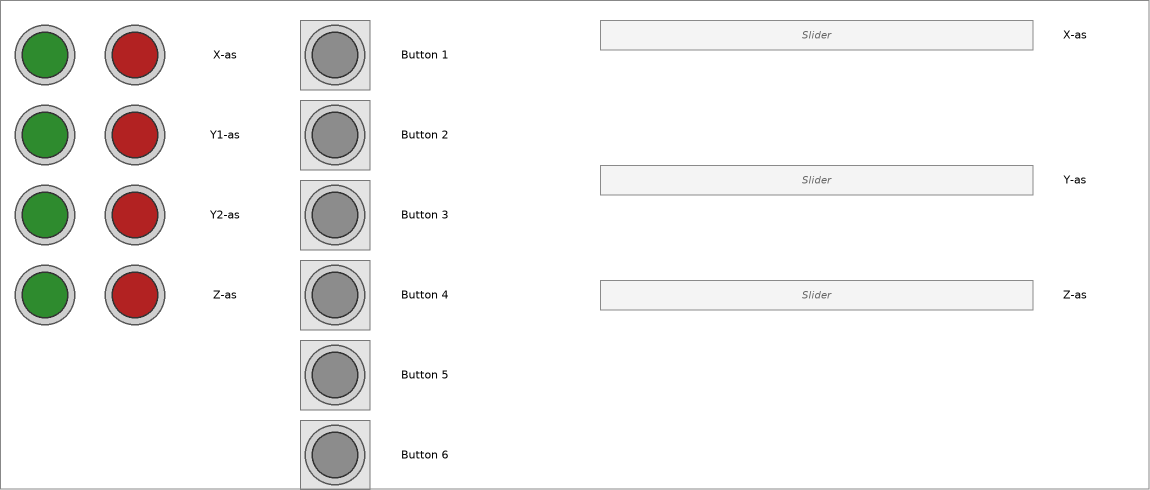
VISUALIZATION Visu  // 1150x490
    Slider (600,20 433x30), variable: GVL.slider1, scale 25..375
    Slider (600,165 433x30), variable: GVL.slider2, scale 25..375
    Slider (600,280 433x30), variable: GVL.slider3, scale 25..125
    Lamp1 (100,20 70x70), variable: GVL.bLed_Rd1, style: Lamp-Lamp1-Red
    Lamp1 (100,260 70x70), variable: GVL.bLed_Rd4, style: Lamp-Lamp1-Red
    Lamp1 (100,180 70x70), variable: GVL.bLed_Rd3, style: Lamp-Lamp1-Red
    Lamp1 (100,100 70x70), variable: GVL.bLed_Rd2, style: Lamp-Lamp1-Red
    Lamp1 (10,180 70x70), variable: GVL.bLed_Gn3, style: Lamp-Lamp1-Green
    Lamp1 (10,100 70x70), variable: GVL.bLed_Gn2, style: Lamp-Lamp1-Green
    Lamp1 (10,260 70x70), variable: GVL.bLed_Gn4, style: Lamp-Lamp1-Green
    Lamp1 (10,20 70x70), variable: GVL.bLed_Gn1, style: Lamp-Lamp1-Green
    Label (150,40 150x30), "X-as"
    Label (150,200 150x30), "Y2-as"
    Label (150,120 150x30), "Y1-as"
    Label (150,280 150x30), "Z-as"
    Label (1000,20 150x30), "X-as"
    Label (1000,165 150x30), "Y-as"
    Label (1000,280 150x30), "Z-as"
    PushSwitch (300,20 70x70), variable: GVL.bButton1, behaviour: TOGGLE, style: Switch-PushSwitch-Gray
    PushSwitch (300,100 70x70), variable: GVL.bButton2, behaviour: TOGGLE, style: Switch-PushSwitch-Gray
    PushSwitch (300,180 70x70), variable: GVL.bButton3, behaviour: TOGGLE, style: Switch-PushSwitch-Gray
    PushSwitch (300,260 70x70), variable: GVL.bButton4, behaviour: TOGGLE, style: Switch-PushSwitch-Gray
    PushSwitch (300,340 70x70), variable: GVL.bButton5, behaviour: TOGGLE, style: Switch-PushSwitch-Gray
    PushSwitch (300,420 70x70), variable: GVL.bButton6, behaviour: TOGGLE, style: Switch-PushSwitch-Gray
    Label (350,40 150x30), "Button 1"
    Label (350,120 150x30), "Button 2"
    Label (350,200 150x30), "Button 3"
    Label (350,280 150x30), "Button 4"
    Label (350,360 150x30), "Button 5"
    Label (350,440 150x30), "Button 6"
END_VISUALIZATION

(* stored: Version 1.1.0.1, ProductVersion 3.1.4026.8
   Visu Visu: Id {7ac9aaa2-04e4-4569-95cf-414302cdea46} *)
